FUNCTION_BLOCK NumberSelection
  (* Standard: 61499-2 *)
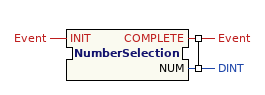
  EVENT_INPUT
    INIT;
  END_EVENT
  EVENT_OUTPUT
    COMPLETE WITH NUM;
  END_EVENT
  VAR_OUTPUT
    NUM : DINT;
  END_VAR
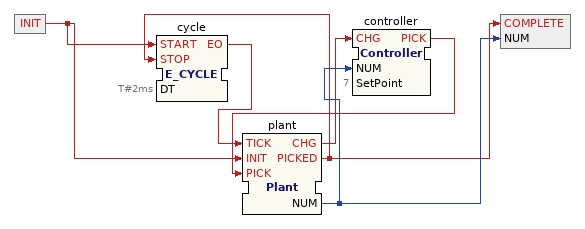
  FBS
    plant : Plant;
    controller : Controller(SetPoint := 7);
    cycle : E_CYCLE(DT := T#2ms);
  END_FBS
  EVENT_CONNECTIONS
    cycle.EO TO plant.TICK;
    INIT TO cycle.START;
    INIT TO plant.INIT;
    plant.CHG TO controller.CHG;
    controller.PICK TO plant.PICK;
    plant.PICKED TO COMPLETE;
    plant.PICKED TO cycle.STOP;
  END_CONNECTIONS
  DATA_CONNECTIONS
    plant.NUM TO controller.NUM;
    plant.NUM TO NUM;
  END_CONNECTIONS
END_FUNCTION_BLOCK
